% RSLogix 500 project I2P PROJECT 01 - TANK 1 TEMPLATE_BAK048.RSS, saved by version 10.00.00.00 %
PROJECT "UNTITLED"    % processor: Bul.1763 MicroLogix 1100 Series B %

PROGRAM FILES
  LAD 2 "MAIN"  6 rungs  % Process Tank 1 Controls %
  LAD 3 "SIM"  18 rungs  % Simulation %
  LAD 4 "ERR"  6 rungs  % Error Flasher %

DATA FILES
  O0 OUTPUT  4 elements
  I1 INPUT  6 elements
  S2 STATUS  66 elements
  B3 BINARY  11 elements
  T4 TIMER  17 elements
  C5 COUNTER  11 elements
  R6 CONTROL  1 elements
  N7 INTEGER  11 elements
  F8 FLOAT  2 elements

LADDER 2 "MAIN"    % Process Tank 1 Controls %
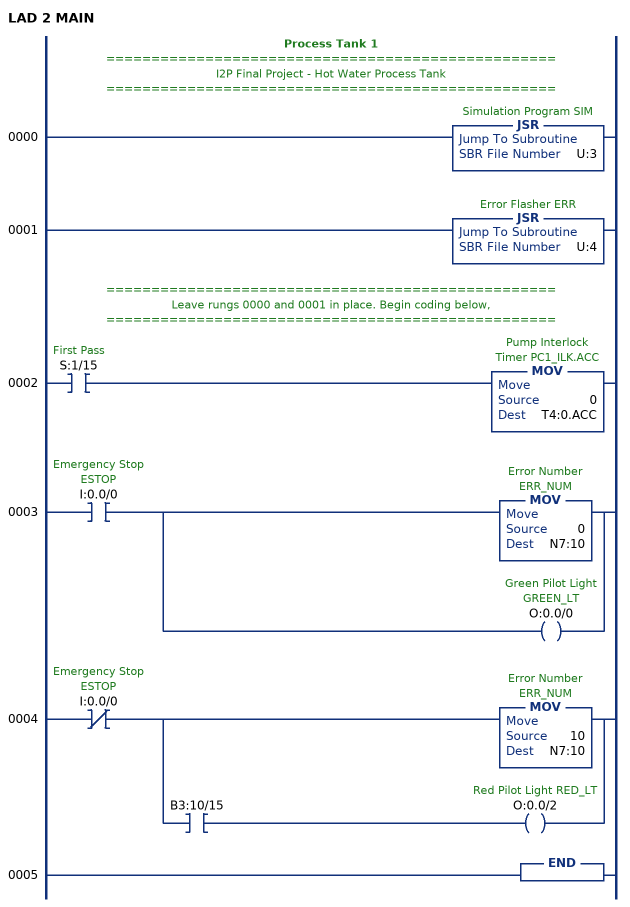
% Rung: 0 %
% TITLE: Process Tank 1 %
% ==================================================
%   I2P Final Project - Hot Water Process Tank
% ================================================== %
SOR JSR U:3 EOR
%   U:3  SIM  "Simulation Program" %
% Rung: 1 %
SOR JSR U:4 EOR
%   U:4  ERR  "Error Flasher" %
% Rung: 2 %
% ==================================================
%    Leave rungs 0000 and 0001 in place. Begin coding below,
% ================================================== %
SOR XIC S:1/15 MOV 0 T4:0.ACC EOR
%   S:1/15  "First Pass" %
%   T4:0  PC1_ILK  "Pump Interlock Timer" %
% Rung: 3 %
SOR XIC I:0.0/0 BST MOV 0 N7:10 NXB OTE O:0.0/0 BND EOR
%   I:0.0/0  ESTOP  "Emergency Stop" %
%   N7:10  ERR_NUM  "Error Number" %
%   O:0.0/0  GREEN_LT  "Green Pilot Light" %
% Rung: 4 %
SOR XIO I:0.0/0 BST MOV 10 N7:10 NXB XIC B3:10/15 OTE O:0.0/2 BND EOR
%   I:0.0/0  ESTOP  "Emergency Stop" %
%   N7:10  ERR_NUM  "Error Number" %
%   O:0.0/2  RED_LT  "Red Pilot Light" %
% Rung: 5 %
SOR END EOR

LADDER 3 "SIM"    % Simulation %
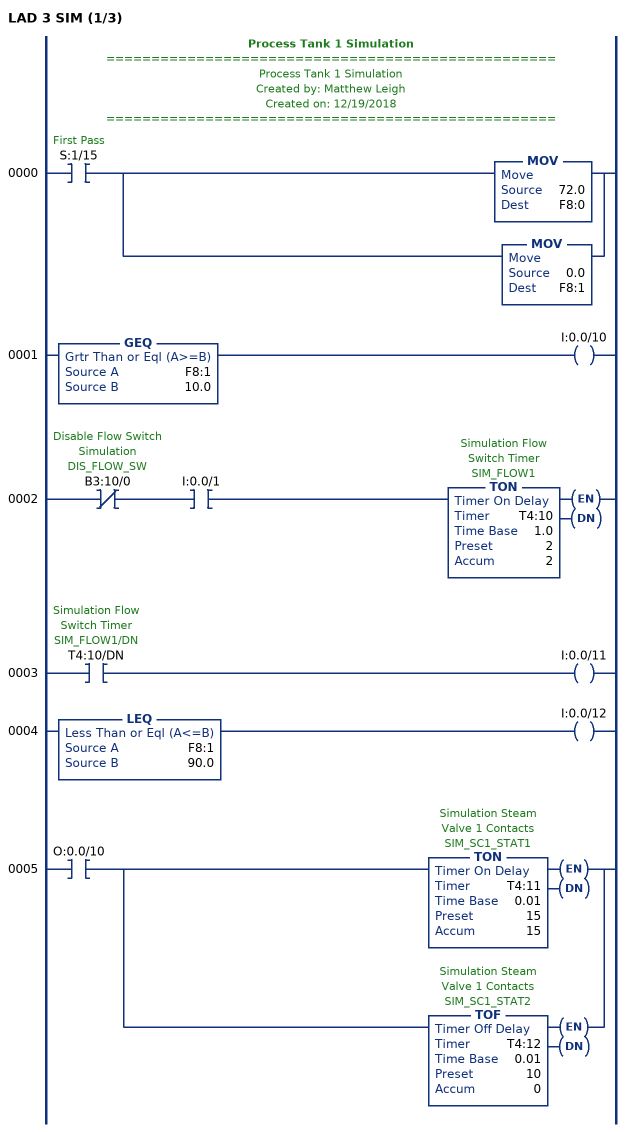
% Rung: 0 %
% TITLE: Process Tank 1 Simulation %
% ==================================================
%      Process Tank 1 Simulation
%      Created by: Matthew Leigh
%      Created on: 12/19/2018
% ================================================== %
SOR XIC S:1/15 BST MOV 72.0 F8:0 NXB MOV 0.0 F8:1 BND EOR
%   S:1/15  "First Pass" %
% Rung: 1 %
SOR GEQ F8:1 10.0 OTE I:0.0/10 EOR
% Rung: 2 %
SOR XIO B3:10/0 XIC I:0.0/1 TON T4:10 1.0 2 2 EOR
%   B3:10/0  DIS_FLOW_SW  "Disable Flow Switch Simulation" %
%   T4:10  SIM_FLOW1  "Simulation Flow Switch Timer" %
% Rung: 3 %
SOR XIC T4:10/DN OTE I:0.0/11 EOR
%   T4:10  SIM_FLOW1  "Simulation Flow Switch Timer" %
% Rung: 4 %
SOR LEQ F8:1 90.0 OTE I:0.0/12 EOR
% Rung: 5 %
SOR XIC O:0.0/10 BST TON T4:11 0.01 15 15 NXB TOF T4:12 0.01 10 0 BND EOR
%   T4:11  SIM_SC1_STAT1  "Simulation Steam Valve 1 Contacts" %
%   T4:12  SIM_SC1_STAT2  "Simulation Steam Valve 1 Contacts" %

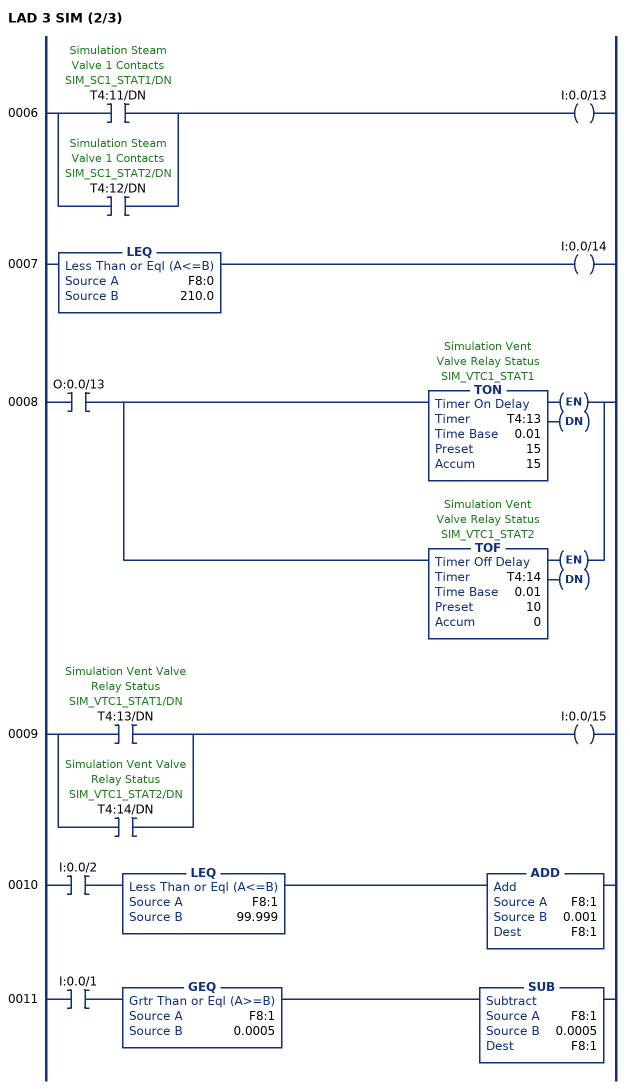
% Rung: 6 %
SOR BST XIC T4:11/DN NXB XIC T4:12/DN BND OTE I:0.0/13 EOR
%   T4:11  SIM_SC1_STAT1  "Simulation Steam Valve 1 Contacts" %
%   T4:12  SIM_SC1_STAT2  "Simulation Steam Valve 1 Contacts" %
% Rung: 7 %
SOR LEQ F8:0 210.0 OTE I:0.0/14 EOR
% Rung: 8 %
SOR XIC O:0.0/13 BST TON T4:13 0.01 15 15 NXB TOF T4:14 0.01 10 0 BND EOR
%   T4:13  SIM_VTC1_STAT1  "Simulation Vent Valve Relay Status" %
%   T4:14  SIM_VTC1_STAT2  "Simulation Vent Valve Relay Status" %
% Rung: 9 %
SOR BST XIC T4:13/DN NXB XIC T4:14/DN BND OTE I:0.0/15 EOR
%   T4:13  SIM_VTC1_STAT1  "Simulation Vent Valve Relay Status" %
%   T4:14  SIM_VTC1_STAT2  "Simulation Vent Valve Relay Status" %
% Rung: 10 %
SOR XIC I:0.0/2 LEQ F8:1 99.999 ADD F8:1 0.001 F8:1 EOR
% Rung: 11 %
SOR XIC I:0.0/1 GEQ F8:1 0.0005 SUB F8:1 0.0005 F8:1 EOR

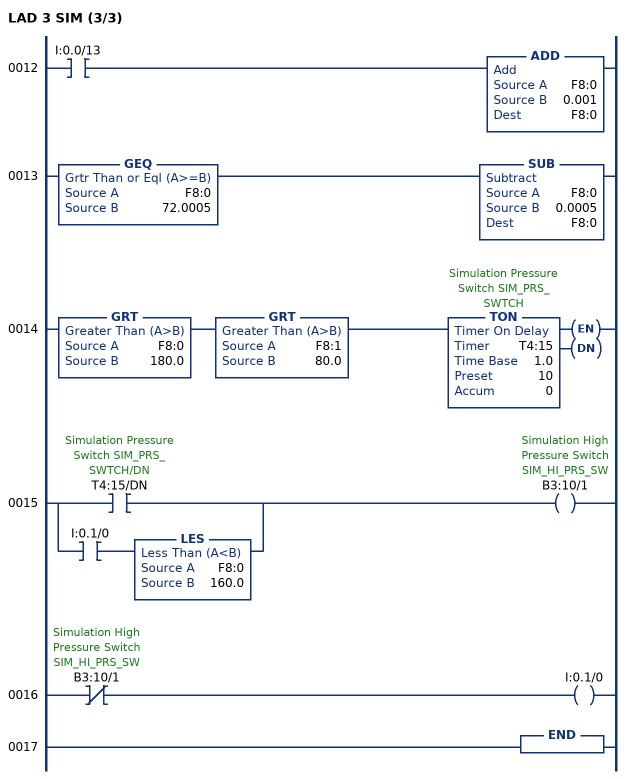
% Rung: 12 %
SOR XIC I:0.0/13 ADD F8:0 0.001 F8:0 EOR
% Rung: 13 %
SOR GEQ F8:0 72.0005 SUB F8:0 0.0005 F8:0 EOR
% Rung: 14 %
SOR GRT F8:0 180.0 GRT F8:1 80.0 TON T4:15 1.0 10 0 EOR
%   T4:15  SIM_PRS_SWTCH  "Simulation Pressure Switch" %
% Rung: 15 %
SOR BST XIC T4:15/DN NXB XIC I:0.1/0 LES F8:0 160.0 BND OTE B3:10/1 EOR
%   T4:15  SIM_PRS_SWTCH  "Simulation Pressure Switch" %
%   B3:10/1  SIM_HI_PRS_SW  "Simulation High Pressure Switch" %
% Rung: 16 %
SOR XIO B3:10/1 OTE I:0.1/0 EOR
%   B3:10/1  SIM_HI_PRS_SW  "Simulation High Pressure Switch" %
% Rung: 17 %
SOR END EOR

LADDER 4 "ERR"    % Error Flasher %
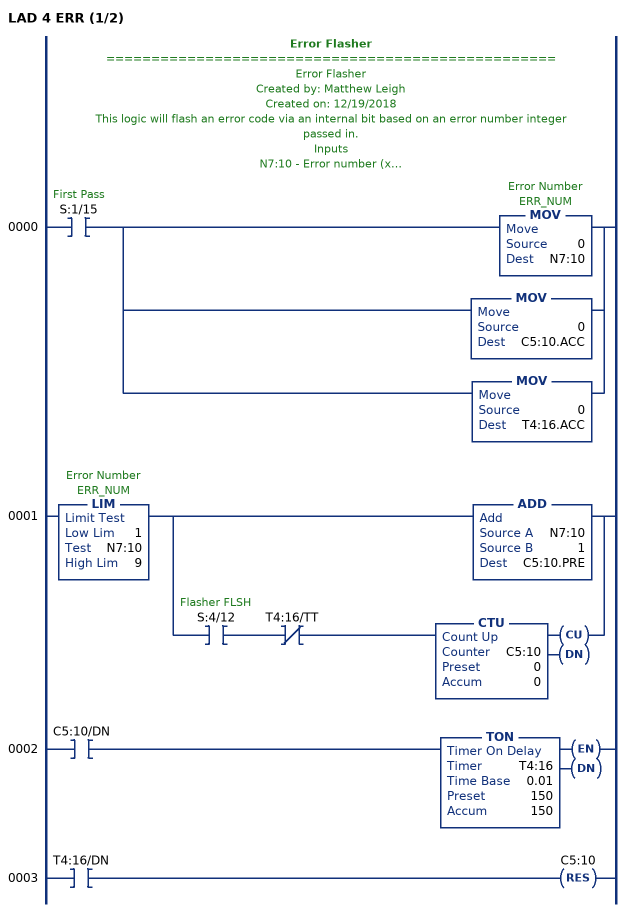
% Rung: 0 %
% TITLE: Error Flasher %
% ==================================================
%      Error Flasher
%      Created by: Matthew Leigh
%      Created on: 12/19/2018
% 
%      This logic will flash an error code via an internal bit based on an error number integer passed in.
% 
%      Inputs
%         N7:10 - Error number (x)
%            x < 0                  Flash Slowly
%            0 < x < 10          Flash Number
%            x = 10                Flash Fast
%            x = 0 or x > 10   On Solid
% 
%      Outputs
%         B3:10/15 - Flashing bit
% 
% ================================================== %
SOR XIC S:1/15 BST MOV 0 N7:10 NXB MOV 0 C5:10.ACC NXB MOV 0 T4:16.ACC BND EOR
%   S:1/15  "First Pass" %
%   N7:10  ERR_NUM  "Error Number" %
% Rung: 1 %
SOR LIM 1 N7:10 9 BST ADD N7:10 1 C5:10.PRE NXB XIC S:4/12 XIO T4:16/TT CTU C5:10 0 0 BND EOR
%   N7:10  ERR_NUM  "Error Number" %
%   S:4/12  FLSH  "Flasher" %
% Rung: 2 %
SOR XIC C5:10/DN TON T4:16 0.01 150 150 EOR
% Rung: 3 %
SOR XIC T4:16/DN RES C5:10 EOR

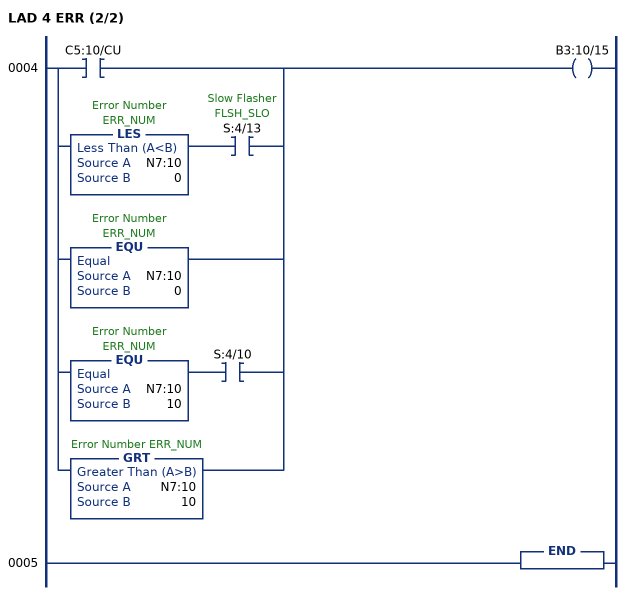
% Rung: 4 %
SOR BST XIC C5:10/CU NXB LES N7:10 0 XIC S:4/13 NXB EQU N7:10 0 NXB EQU N7:10 10 XIC S:4/10 NXB GRT N7:10 10 BND OTE B3:10/15 EOR
%   N7:10  ERR_NUM  "Error Number" %
%   S:4/13  FLSH_SLO  "Slow Flasher" %
% Rung: 5 %
SOR END EOR

OTHER DOCUMENTED ADDRESSES
  S:4/11  FLSH_FST  "Fast Flasher"

DATA TABLE (non-zero values as saved)
DATA B3
% B3:10 % 0X8000
DATA T4
% .PRE .ACC %
% T4:0 % 5 0
% T4:10 % 2 2
% T4:11 % 15 15
% T4:12 % 10 0
% T4:13 % 15 15
% T4:14 % 10 0
% T4:15 % 10 0
% T4:16 % 150 150
DATA F8
% F8:0 % 136.7956 0
